Fanuc TP program (LS listing): MOTIONPROBE.LS

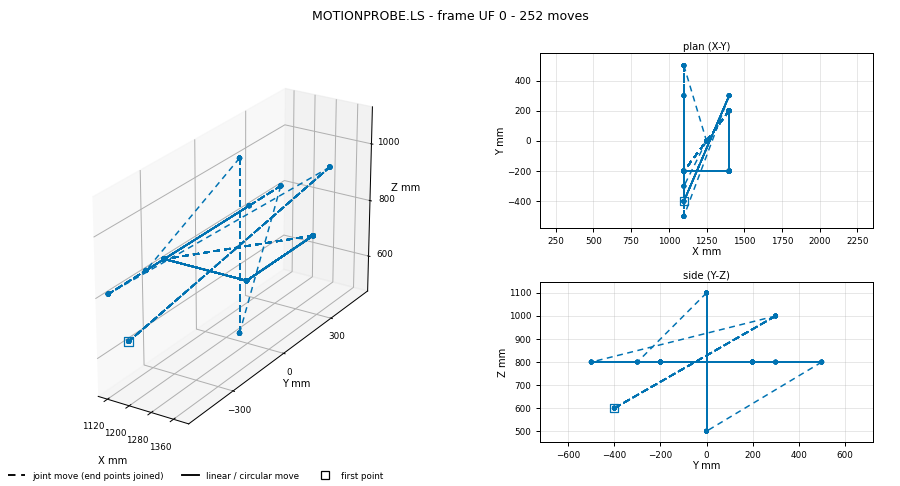
[picture p0: tool path of MOTIONPROBE.LS in frame UF 0, 252 of 252 moves have a stored position in this frame; points joined in program order, loops and branches not executed]
/PROG  MOTIONPROBE
/ATTR
OWNER		= MNEDITOR;
COMMENT		= "motion probe";
PROG_SIZE	= 0;
CREATE		= DATE 26-01-01  TIME 00:00:00;
MODIFIED	= DATE 26-01-01  TIME 00:00:00;
FILE_NAME	= ;
VERSION		= 0;
LINE_COUNT	= 737;
MEMORY_SIZE	= 0;
PROTECT		= READ_WRITE;
TCD:  STACK_SIZE	= 0,
      TASK_PRIORITY	= 50,
      TIME_SLICE	= 0,
      BUSY_LAMP_OFF	= 0,
      ABORT_REQUEST	= 0,
      PAUSE_REQUEST	= 0;
DEFAULT_GROUP	= 1,*,*,*,*;
CONTROL_CODE	= 00000000 00000000;
/MN
   1:  !CrossArm motion probe ;
   2:  PR[20]=P[12]    ;
   3:  UTOOL[1]=PR[20] ;
   4:  UFRAME_NUM=0 ;
   5:  UTOOL_NUM=1 ;
   6:  !joint 5% ;
   7:J P[6] 30% FINE    ;
   8:  TIMER[1]=RESET ;
   9:  TIMER[1]=START ;
  10:J P[7] 5% FINE    ;
  11:  TIMER[1]=STOP ;
  12:  R[101]=TIMER[1]    ;
  13:  !joint 10% ;
  14:J P[6] 30% FINE    ;
  15:  TIMER[1]=RESET ;
  16:  TIMER[1]=START ;
  17:J P[7] 10% FINE    ;
  18:  TIMER[1]=STOP ;
  19:  R[102]=TIMER[1]    ;
  20:  !joint 15% ;
  21:J P[6] 30% FINE    ;
  22:  TIMER[1]=RESET ;
  23:  TIMER[1]=START ;
  24:J P[7] 15% FINE    ;
  25:  TIMER[1]=STOP ;
  26:  R[103]=TIMER[1]    ;
  27:  !joint 20% ;
  28:J P[6] 30% FINE    ;
  29:  TIMER[1]=RESET ;
  30:  TIMER[1]=START ;
  31:J P[7] 20% FINE    ;
  32:  TIMER[1]=STOP ;
  33:  R[104]=TIMER[1]    ;
  34:  !joint 25% ;
  35:J P[6] 30% FINE    ;
  36:  TIMER[1]=RESET ;
  37:  TIMER[1]=START ;
  38:J P[7] 25% FINE    ;
  39:  TIMER[1]=STOP ;
  40:  R[105]=TIMER[1]    ;
  41:  !joint 30% ;
  42:J P[6] 30% FINE    ;
  43:  TIMER[1]=RESET ;
  44:  TIMER[1]=START ;
  45:J P[7] 30% FINE    ;
  46:  TIMER[1]=STOP ;
  47:  R[106]=TIMER[1]    ;
  48:  !joint 40% ;
  49:J P[6] 30% FINE    ;
  50:  TIMER[1]=RESET ;
  51:  TIMER[1]=START ;
  52:J P[7] 40% FINE    ;
  53:  TIMER[1]=STOP ;
  54:  R[107]=TIMER[1]    ;
  55:  !joint 50% ;
  56:J P[6] 30% FINE    ;
  57:  TIMER[1]=RESET ;
  58:  TIMER[1]=START ;
  59:J P[7] 50% FINE    ;
  60:  TIMER[1]=STOP ;
  61:  R[108]=TIMER[1]    ;
  62:  !joint 70% ;
  63:J P[6] 30% FINE    ;
  64:  TIMER[1]=RESET ;
  65:  TIMER[1]=START ;
  66:J P[7] 70% FINE    ;
  67:  TIMER[1]=STOP ;
  68:  R[109]=TIMER[1]    ;
  69:  !joint 100% ;
  70:J P[6] 30% FINE    ;
  71:  TIMER[1]=RESET ;
  72:  TIMER[1]=START ;
  73:J P[7] 100% FINE    ;
  74:  TIMER[1]=STOP ;
  75:  R[110]=TIMER[1]    ;
  76:  !swing 5% ;
  77:J P[8] 30% FINE    ;
  78:  TIMER[1]=RESET ;
  79:  TIMER[1]=START ;
  80:J P[9] 5% FINE    ;
  81:  TIMER[1]=STOP ;
  82:  R[111]=TIMER[1]    ;
  83:  !swing 10% ;
  84:J P[8] 30% FINE    ;
  85:  TIMER[1]=RESET ;
  86:  TIMER[1]=START ;
  87:J P[9] 10% FINE    ;
  88:  TIMER[1]=STOP ;
  89:  R[112]=TIMER[1]    ;
  90:  !swing 15% ;
  91:J P[8] 30% FINE    ;
  92:  TIMER[1]=RESET ;
  93:  TIMER[1]=START ;
  94:J P[9] 15% FINE    ;
  95:  TIMER[1]=STOP ;
  96:  R[113]=TIMER[1]    ;
  97:  !swing 20% ;
  98:J P[8] 30% FINE    ;
  99:  TIMER[1]=RESET ;
 100:  TIMER[1]=START ;
 101:J P[9] 20% FINE    ;
 102:  TIMER[1]=STOP ;
 103:  R[114]=TIMER[1]    ;
 104:  !swing 25% ;
 105:J P[8] 30% FINE    ;
 106:  TIMER[1]=RESET ;
 107:  TIMER[1]=START ;
 108:J P[9] 25% FINE    ;
 109:  TIMER[1]=STOP ;
 110:  R[115]=TIMER[1]    ;
 111:  !swing 30% ;
 112:J P[8] 30% FINE    ;
 113:  TIMER[1]=RESET ;
 114:  TIMER[1]=START ;
 115:J P[9] 30% FINE    ;
 116:  TIMER[1]=STOP ;
 117:  R[116]=TIMER[1]    ;
 118:  !swing 40% ;
 119:J P[8] 30% FINE    ;
 120:  TIMER[1]=RESET ;
 121:  TIMER[1]=START ;
 122:J P[9] 40% FINE    ;
 123:  TIMER[1]=STOP ;
 124:  R[117]=TIMER[1]    ;
 125:  !swing 50% ;
 126:J P[8] 30% FINE    ;
 127:  TIMER[1]=RESET ;
 128:  TIMER[1]=START ;
 129:J P[9] 50% FINE    ;
 130:  TIMER[1]=STOP ;
 131:  R[118]=TIMER[1]    ;
 132:  !swing 70% ;
 133:J P[8] 30% FINE    ;
 134:  TIMER[1]=RESET ;
 135:  TIMER[1]=START ;
 136:J P[9] 70% FINE    ;
 137:  TIMER[1]=STOP ;
 138:  R[119]=TIMER[1]    ;
 139:  !swing 100% ;
 140:J P[8] 30% FINE    ;
 141:  TIMER[1]=RESET ;
 142:  TIMER[1]=START ;
 143:J P[9] 100% FINE    ;
 144:  TIMER[1]=STOP ;
 145:  R[120]=TIMER[1]    ;
 146:  !rise 5% ;
 147:J P[10] 30% FINE    ;
 148:  TIMER[1]=RESET ;
 149:  TIMER[1]=START ;
 150:J P[11] 5% FINE    ;
 151:  TIMER[1]=STOP ;
 152:  R[121]=TIMER[1]    ;
 153:  !rise 10% ;
 154:J P[10] 30% FINE    ;
 155:  TIMER[1]=RESET ;
 156:  TIMER[1]=START ;
 157:J P[11] 10% FINE    ;
 158:  TIMER[1]=STOP ;
 159:  R[122]=TIMER[1]    ;
 160:  !rise 15% ;
 161:J P[10] 30% FINE    ;
 162:  TIMER[1]=RESET ;
 163:  TIMER[1]=START ;
 164:J P[11] 15% FINE    ;
 165:  TIMER[1]=STOP ;
 166:  R[123]=TIMER[1]    ;
 167:  !rise 20% ;
 168:J P[10] 30% FINE    ;
 169:  TIMER[1]=RESET ;
 170:  TIMER[1]=START ;
 171:J P[11] 20% FINE    ;
 172:  TIMER[1]=STOP ;
 173:  R[124]=TIMER[1]    ;
 174:  !rise 25% ;
 175:J P[10] 30% FINE    ;
 176:  TIMER[1]=RESET ;
 177:  TIMER[1]=START ;
 178:J P[11] 25% FINE    ;
 179:  TIMER[1]=STOP ;
 180:  R[125]=TIMER[1]    ;
 181:  !rise 30% ;
 182:J P[10] 30% FINE    ;
 183:  TIMER[1]=RESET ;
 184:  TIMER[1]=START ;
 185:J P[11] 30% FINE    ;
 186:  TIMER[1]=STOP ;
 187:  R[126]=TIMER[1]    ;
 188:  !rise 40% ;
 189:J P[10] 30% FINE    ;
 190:  TIMER[1]=RESET ;
 191:  TIMER[1]=START ;
 192:J P[11] 40% FINE    ;
 193:  TIMER[1]=STOP ;
 194:  R[127]=TIMER[1]    ;
 195:  !rise 50% ;
 196:J P[10] 30% FINE    ;
 197:  TIMER[1]=RESET ;
 198:  TIMER[1]=START ;
 199:J P[11] 50% FINE    ;
 200:  TIMER[1]=STOP ;
 201:  R[128]=TIMER[1]    ;
 202:  !rise 70% ;
 203:J P[10] 30% FINE    ;
 204:  TIMER[1]=RESET ;
 205:  TIMER[1]=START ;
 206:J P[11] 70% FINE    ;
 207:  TIMER[1]=STOP ;
 208:  R[129]=TIMER[1]    ;
 209:  !rise 100% ;
 210:J P[10] 30% FINE    ;
 211:  TIMER[1]=RESET ;
 212:  TIMER[1]=START ;
 213:J P[11] 100% FINE    ;
 214:  TIMER[1]=STOP ;
 215:  R[130]=TIMER[1]    ;
 216:  !linear 100mm/sec ;
 217:J P[4] 30% FINE    ;
 218:  TIMER[1]=RESET ;
 219:  TIMER[1]=START ;
 220:L P[5] 100mm/sec FINE    ;
 221:  TIMER[1]=STOP ;
 222:  R[131]=TIMER[1]    ;
 223:  !linear 200mm/sec ;
 224:J P[4] 30% FINE    ;
 225:  TIMER[1]=RESET ;
 226:  TIMER[1]=START ;
 227:L P[5] 200mm/sec FINE    ;
 228:  TIMER[1]=STOP ;
 229:  R[132]=TIMER[1]    ;
 230:  !linear 500mm/sec ;
 231:J P[4] 30% FINE    ;
 232:  TIMER[1]=RESET ;
 233:  TIMER[1]=START ;
 234:L P[5] 500mm/sec FINE    ;
 235:  TIMER[1]=STOP ;
 236:  R[133]=TIMER[1]    ;
 237:  !linear 1000mm/sec ;
 238:J P[4] 30% FINE    ;
 239:  TIMER[1]=RESET ;
 240:  TIMER[1]=START ;
 241:L P[5] 1000mm/sec FINE    ;
 242:  TIMER[1]=STOP ;
 243:  R[134]=TIMER[1]    ;
 244:  !linear 1500mm/sec ;
 245:J P[4] 30% FINE    ;
 246:  TIMER[1]=RESET ;
 247:  TIMER[1]=START ;
 248:L P[5] 1500mm/sec FINE    ;
 249:  TIMER[1]=STOP ;
 250:  R[135]=TIMER[1]    ;
 251:  !linear 2000mm/sec ;
 252:J P[4] 30% FINE    ;
 253:  TIMER[1]=RESET ;
 254:  TIMER[1]=START ;
 255:L P[5] 2000mm/sec FINE    ;
 256:  TIMER[1]=STOP ;
 257:  R[136]=TIMER[1]    ;
 258:  !corner 200mm/sec FINE ;
 259:J P[1] 30% FINE    ;
 260:  TIMER[1]=RESET ;
 261:  TIMER[1]=START ;
 262:L P[2] 200mm/sec FINE    ;
 263:L P[3] 200mm/sec FINE    ;
 264:  TIMER[1]=STOP ;
 265:  R[137]=TIMER[1]    ;
 266:  !corner 200mm/sec CNT0 ;
 267:J P[1] 30% FINE    ;
 268:  TIMER[1]=RESET ;
 269:  TIMER[1]=START ;
 270:L P[2] 200mm/sec CNT0    ;
 271:L P[3] 200mm/sec FINE    ;
 272:  TIMER[1]=STOP ;
 273:  R[138]=TIMER[1]    ;
 274:  !corner 200mm/sec CNT10 ;
 275:J P[1] 30% FINE    ;
 276:  TIMER[1]=RESET ;
 277:  TIMER[1]=START ;
 278:L P[2] 200mm/sec CNT10    ;
 279:L P[3] 200mm/sec FINE    ;
 280:  TIMER[1]=STOP ;
 281:  R[139]=TIMER[1]    ;
 282:  !corner 200mm/sec CNT20 ;
 283:J P[1] 30% FINE    ;
 284:  TIMER[1]=RESET ;
 285:  TIMER[1]=START ;
 286:L P[2] 200mm/sec CNT20    ;
 287:L P[3] 200mm/sec FINE    ;
 288:  TIMER[1]=STOP ;
 289:  R[140]=TIMER[1]    ;
 290:  !corner 200mm/sec CNT30 ;
 291:J P[1] 30% FINE    ;
 292:  TIMER[1]=RESET ;
 293:  TIMER[1]=START ;
 294:L P[2] 200mm/sec CNT30    ;
 295:L P[3] 200mm/sec FINE    ;
 296:  TIMER[1]=STOP ;
 297:  R[141]=TIMER[1]    ;
 298:  !corner 200mm/sec CNT40 ;
 299:J P[1] 30% FINE    ;
 300:  TIMER[1]=RESET ;
 301:  TIMER[1]=START ;
 302:L P[2] 200mm/sec CNT40    ;
 303:L P[3] 200mm/sec FINE    ;
 304:  TIMER[1]=STOP ;
 305:  R[142]=TIMER[1]    ;
 306:  !corner 200mm/sec CNT50 ;
 307:J P[1] 30% FINE    ;
 308:  TIMER[1]=RESET ;
 309:  TIMER[1]=START ;
 310:L P[2] 200mm/sec CNT50    ;
 311:L P[3] 200mm/sec FINE    ;
 312:  TIMER[1]=STOP ;
 313:  R[143]=TIMER[1]    ;
 314:  !corner 200mm/sec CNT60 ;
 315:J P[1] 30% FINE    ;
 316:  TIMER[1]=RESET ;
 317:  TIMER[1]=START ;
 318:L P[2] 200mm/sec CNT60    ;
 319:L P[3] 200mm/sec FINE    ;
 320:  TIMER[1]=STOP ;
 321:  R[144]=TIMER[1]    ;
 322:  !corner 200mm/sec CNT70 ;
 323:J P[1] 30% FINE    ;
 324:  TIMER[1]=RESET ;
 325:  TIMER[1]=START ;
 326:L P[2] 200mm/sec CNT70    ;
 327:L P[3] 200mm/sec FINE    ;
 328:  TIMER[1]=STOP ;
 329:  R[145]=TIMER[1]    ;
 330:  !corner 200mm/sec CNT80 ;
 331:J P[1] 30% FINE    ;
 332:  TIMER[1]=RESET ;
 333:  TIMER[1]=START ;
 334:L P[2] 200mm/sec CNT80    ;
 335:L P[3] 200mm/sec FINE    ;
 336:  TIMER[1]=STOP ;
 337:  R[146]=TIMER[1]    ;
 338:  !corner 200mm/sec CNT90 ;
 339:J P[1] 30% FINE    ;
 340:  TIMER[1]=RESET ;
 341:  TIMER[1]=START ;
 342:L P[2] 200mm/sec CNT90    ;
 343:L P[3] 200mm/sec FINE    ;
 344:  TIMER[1]=STOP ;
 345:  R[147]=TIMER[1]    ;
 346:  !corner 200mm/sec CNT100 ;
 347:J P[1] 30% FINE    ;
 348:  TIMER[1]=RESET ;
 349:  TIMER[1]=START ;
 350:L P[2] 200mm/sec CNT100    ;
 351:L P[3] 200mm/sec FINE    ;
 352:  TIMER[1]=STOP ;
 353:  R[148]=TIMER[1]    ;
 354:  !corner 500mm/sec FINE ;
 355:J P[1] 30% FINE    ;
 356:  TIMER[1]=RESET ;
 357:  TIMER[1]=START ;
 358:L P[2] 500mm/sec FINE    ;
 359:L P[3] 500mm/sec FINE    ;
 360:  TIMER[1]=STOP ;
 361:  R[149]=TIMER[1]    ;
 362:  !corner 500mm/sec CNT0 ;
 363:J P[1] 30% FINE    ;
 364:  TIMER[1]=RESET ;
 365:  TIMER[1]=START ;
 366:L P[2] 500mm/sec CNT0    ;
 367:L P[3] 500mm/sec FINE    ;
 368:  TIMER[1]=STOP ;
 369:  R[150]=TIMER[1]    ;
 370:  !corner 500mm/sec CNT10 ;
 371:J P[1] 30% FINE    ;
 372:  TIMER[1]=RESET ;
 373:  TIMER[1]=START ;
 374:L P[2] 500mm/sec CNT10    ;
 375:L P[3] 500mm/sec FINE    ;
 376:  TIMER[1]=STOP ;
 377:  R[151]=TIMER[1]    ;
 378:  !corner 500mm/sec CNT20 ;
 379:J P[1] 30% FINE    ;
 380:  TIMER[1]=RESET ;
 381:  TIMER[1]=START ;
 382:L P[2] 500mm/sec CNT20    ;
 383:L P[3] 500mm/sec FINE    ;
 384:  TIMER[1]=STOP ;
 385:  R[152]=TIMER[1]    ;
 386:  !corner 500mm/sec CNT30 ;
 387:J P[1] 30% FINE    ;
 388:  TIMER[1]=RESET ;
 389:  TIMER[1]=START ;
 390:L P[2] 500mm/sec CNT30    ;
 391:L P[3] 500mm/sec FINE    ;
 392:  TIMER[1]=STOP ;
 393:  R[153]=TIMER[1]    ;
 394:  !corner 500mm/sec CNT40 ;
 395:J P[1] 30% FINE    ;
 396:  TIMER[1]=RESET ;
 397:  TIMER[1]=START ;
 398:L P[2] 500mm/sec CNT40    ;
 399:L P[3] 500mm/sec FINE    ;
 400:  TIMER[1]=STOP ;
 401:  R[154]=TIMER[1]    ;
 402:  !corner 500mm/sec CNT50 ;
 403:J P[1] 30% FINE    ;
 404:  TIMER[1]=RESET ;
 405:  TIMER[1]=START ;
 406:L P[2] 500mm/sec CNT50    ;
 407:L P[3] 500mm/sec FINE    ;
 408:  TIMER[1]=STOP ;
 409:  R[155]=TIMER[1]    ;
 410:  !corner 500mm/sec CNT60 ;
 411:J P[1] 30% FINE    ;
 412:  TIMER[1]=RESET ;
 413:  TIMER[1]=START ;
 414:L P[2] 500mm/sec CNT60    ;
 415:L P[3] 500mm/sec FINE    ;
 416:  TIMER[1]=STOP ;
 417:  R[156]=TIMER[1]    ;
 418:  !corner 500mm/sec CNT70 ;
 419:J P[1] 30% FINE    ;
 420:  TIMER[1]=RESET ;
 421:  TIMER[1]=START ;
 422:L P[2] 500mm/sec CNT70    ;
 423:L P[3] 500mm/sec FINE    ;
 424:  TIMER[1]=STOP ;
 425:  R[157]=TIMER[1]    ;
 426:  !corner 500mm/sec CNT80 ;
 427:J P[1] 30% FINE    ;
 428:  TIMER[1]=RESET ;
 429:  TIMER[1]=START ;
 430:L P[2] 500mm/sec CNT80    ;
 431:L P[3] 500mm/sec FINE    ;
 432:  TIMER[1]=STOP ;
 433:  R[158]=TIMER[1]    ;
 434:  !corner 500mm/sec CNT90 ;
 435:J P[1] 30% FINE    ;
 436:  TIMER[1]=RESET ;
 437:  TIMER[1]=START ;
 438:L P[2] 500mm/sec CNT90    ;
 439:L P[3] 500mm/sec FINE    ;
 440:  TIMER[1]=STOP ;
 441:  R[159]=TIMER[1]    ;
 442:  !corner 500mm/sec CNT100 ;
 443:J P[1] 30% FINE    ;
 444:  TIMER[1]=RESET ;
 445:  TIMER[1]=START ;
 446:L P[2] 500mm/sec CNT100    ;
 447:L P[3] 500mm/sec FINE    ;
 448:  TIMER[1]=STOP ;
 449:  R[160]=TIMER[1]    ;
 450:  !corner 1000mm/sec FINE ;
 451:J P[1] 30% FINE    ;
 452:  TIMER[1]=RESET ;
 453:  TIMER[1]=START ;
 454:L P[2] 1000mm/sec FINE    ;
 455:L P[3] 1000mm/sec FINE    ;
 456:  TIMER[1]=STOP ;
 457:  R[161]=TIMER[1]    ;
 458:  !corner 1000mm/sec CNT0 ;
 459:J P[1] 30% FINE    ;
 460:  TIMER[1]=RESET ;
 461:  TIMER[1]=START ;
 462:L P[2] 1000mm/sec CNT0    ;
 463:L P[3] 1000mm/sec FINE    ;
 464:  TIMER[1]=STOP ;
 465:  R[162]=TIMER[1]    ;
 466:  !corner 1000mm/sec CNT10 ;
 467:J P[1] 30% FINE    ;
 468:  TIMER[1]=RESET ;
 469:  TIMER[1]=START ;
 470:L P[2] 1000mm/sec CNT10    ;
 471:L P[3] 1000mm/sec FINE    ;
 472:  TIMER[1]=STOP ;
 473:  R[163]=TIMER[1]    ;
 474:  !corner 1000mm/sec CNT20 ;
 475:J P[1] 30% FINE    ;
 476:  TIMER[1]=RESET ;
 477:  TIMER[1]=START ;
 478:L P[2] 1000mm/sec CNT20    ;
 479:L P[3] 1000mm/sec FINE    ;
 480:  TIMER[1]=STOP ;
 481:  R[164]=TIMER[1]    ;
 482:  !corner 1000mm/sec CNT30 ;
 483:J P[1] 30% FINE    ;
 484:  TIMER[1]=RESET ;
 485:  TIMER[1]=START ;
 486:L P[2] 1000mm/sec CNT30    ;
 487:L P[3] 1000mm/sec FINE    ;
 488:  TIMER[1]=STOP ;
 489:  R[165]=TIMER[1]    ;
 490:  !corner 1000mm/sec CNT40 ;
 491:J P[1] 30% FINE    ;
 492:  TIMER[1]=RESET ;
 493:  TIMER[1]=START ;
 494:L P[2] 1000mm/sec CNT40    ;
 495:L P[3] 1000mm/sec FINE    ;
 496:  TIMER[1]=STOP ;
 497:  R[166]=TIMER[1]    ;
 498:  !corner 1000mm/sec CNT50 ;
 499:J P[1] 30% FINE    ;
 500:  TIMER[1]=RESET ;
 501:  TIMER[1]=START ;
 502:L P[2] 1000mm/sec CNT50    ;
 503:L P[3] 1000mm/sec FINE    ;
 504:  TIMER[1]=STOP ;
 505:  R[167]=TIMER[1]    ;
 506:  !corner 1000mm/sec CNT60 ;
 507:J P[1] 30% FINE    ;
 508:  TIMER[1]=RESET ;
 509:  TIMER[1]=START ;
 510:L P[2] 1000mm/sec CNT60    ;
 511:L P[3] 1000mm/sec FINE    ;
 512:  TIMER[1]=STOP ;
 513:  R[168]=TIMER[1]    ;
 514:  !corner 1000mm/sec CNT70 ;
 515:J P[1] 30% FINE    ;
 516:  TIMER[1]=RESET ;
 517:  TIMER[1]=START ;
 518:L P[2] 1000mm/sec CNT70    ;
 519:L P[3] 1000mm/sec FINE    ;
 520:  TIMER[1]=STOP ;
 521:  R[169]=TIMER[1]    ;
 522:  !corner 1000mm/sec CNT80 ;
 523:J P[1] 30% FINE    ;
 524:  TIMER[1]=RESET ;
 525:  TIMER[1]=START ;
 526:L P[2] 1000mm/sec CNT80    ;
 527:L P[3] 1000mm/sec FINE    ;
 528:  TIMER[1]=STOP ;
 529:  R[170]=TIMER[1]    ;
 530:  !corner 1000mm/sec CNT90 ;
 531:J P[1] 30% FINE    ;
 532:  TIMER[1]=RESET ;
 533:  TIMER[1]=START ;
 534:L P[2] 1000mm/sec CNT90    ;
 535:L P[3] 1000mm/sec FINE    ;
 536:  TIMER[1]=STOP ;
 537:  R[171]=TIMER[1]    ;
 538:  !corner 1000mm/sec CNT100 ;
 539:J P[1] 30% FINE    ;
 540:  TIMER[1]=RESET ;
 541:  TIMER[1]=START ;
 542:L P[2] 1000mm/sec CNT100    ;
 543:L P[3] 1000mm/sec FINE    ;
 544:  TIMER[1]=STOP ;
 545:  R[172]=TIMER[1]    ;
 546:  !jcorner 9% FINE ;
 547:J P[1] 30% FINE    ;
 548:  TIMER[1]=RESET ;
 549:  TIMER[1]=START ;
 550:J P[2] 9% FINE    ;
 551:J P[3] 9% FINE    ;
 552:  TIMER[1]=STOP ;
 553:  R[173]=TIMER[1]    ;
 554:  !jcorner 9% CNT0 ;
 555:J P[1] 30% FINE    ;
 556:  TIMER[1]=RESET ;
 557:  TIMER[1]=START ;
 558:J P[2] 9% CNT0    ;
 559:J P[3] 9% FINE    ;
 560:  TIMER[1]=STOP ;
 561:  R[174]=TIMER[1]    ;
 562:  !jcorner 9% CNT10 ;
 563:J P[1] 30% FINE    ;
 564:  TIMER[1]=RESET ;
 565:  TIMER[1]=START ;
 566:J P[2] 9% CNT10    ;
 567:J P[3] 9% FINE    ;
 568:  TIMER[1]=STOP ;
 569:  R[175]=TIMER[1]    ;
 570:  !jcorner 9% CNT20 ;
 571:J P[1] 30% FINE    ;
 572:  TIMER[1]=RESET ;
 573:  TIMER[1]=START ;
 574:J P[2] 9% CNT20    ;
 575:J P[3] 9% FINE    ;
 576:  TIMER[1]=STOP ;
 577:  R[176]=TIMER[1]    ;
 578:  !jcorner 9% CNT30 ;
 579:J P[1] 30% FINE    ;
 580:  TIMER[1]=RESET ;
 581:  TIMER[1]=START ;
 582:J P[2] 9% CNT30    ;
 583:J P[3] 9% FINE    ;
 584:  TIMER[1]=STOP ;
 585:  R[177]=TIMER[1]    ;
 586:  !jcorner 9% CNT40 ;
 587:J P[1] 30% FINE    ;
 588:  TIMER[1]=RESET ;
 589:  TIMER[1]=START ;
 590:J P[2] 9% CNT40    ;
 591:J P[3] 9% FINE    ;
 592:  TIMER[1]=STOP ;
 593:  R[178]=TIMER[1]    ;
 594:  !jcorner 9% CNT50 ;
 595:J P[1] 30% FINE    ;
 596:  TIMER[1]=RESET ;
 597:  TIMER[1]=START ;
 598:J P[2] 9% CNT50    ;
 599:J P[3] 9% FINE    ;
 600:  TIMER[1]=STOP ;
 601:  R[179]=TIMER[1]    ;
 602:  !jcorner 9% CNT60 ;
 603:J P[1] 30% FINE    ;
 604:  TIMER[1]=RESET ;
 605:  TIMER[1]=START ;
 606:J P[2] 9% CNT60    ;
 607:J P[3] 9% FINE    ;
 608:  TIMER[1]=STOP ;
 609:  R[180]=TIMER[1]    ;
 610:  !jcorner 9% CNT70 ;
 611:J P[1] 30% FINE    ;
 612:  TIMER[1]=RESET ;
 613:  TIMER[1]=START ;
 614:J P[2] 9% CNT70    ;
 615:J P[3] 9% FINE    ;
 616:  TIMER[1]=STOP ;
 617:  R[181]=TIMER[1]    ;
 618:  !jcorner 9% CNT80 ;
 619:J P[1] 30% FINE    ;
 620:  TIMER[1]=RESET ;
 621:  TIMER[1]=START ;
 622:J P[2] 9% CNT80    ;
 623:J P[3] 9% FINE    ;
 624:  TIMER[1]=STOP ;
 625:  R[182]=TIMER[1]    ;
 626:  !jcorner 9% CNT90 ;
 627:J P[1] 30% FINE    ;
 628:  TIMER[1]=RESET ;
 629:  TIMER[1]=START ;
 630:J P[2] 9% CNT90    ;
 631:J P[3] 9% FINE    ;
 632:  TIMER[1]=STOP ;
 633:  R[183]=TIMER[1]    ;
 634:  !jcorner 9% CNT100 ;
 635:J P[1] 30% FINE    ;
 636:  TIMER[1]=RESET ;
 637:  TIMER[1]=START ;
 638:J P[2] 9% CNT100    ;
 639:J P[3] 9% FINE    ;
 640:  TIMER[1]=STOP ;
 641:  R[184]=TIMER[1]    ;
 642:  !jcorner 19% FINE ;
 643:J P[1] 30% FINE    ;
 644:  TIMER[1]=RESET ;
 645:  TIMER[1]=START ;
 646:J P[2] 19% FINE    ;
 647:J P[3] 19% FINE    ;
 648:  TIMER[1]=STOP ;
 649:  R[185]=TIMER[1]    ;
 650:  !jcorner 19% CNT0 ;
 651:J P[1] 30% FINE    ;
 652:  TIMER[1]=RESET ;
 653:  TIMER[1]=START ;
 654:J P[2] 19% CNT0    ;
 655:J P[3] 19% FINE    ;
 656:  TIMER[1]=STOP ;
 657:  R[186]=TIMER[1]    ;
 658:  !jcorner 19% CNT10 ;
 659:J P[1] 30% FINE    ;
 660:  TIMER[1]=RESET ;
 661:  TIMER[1]=START ;
 662:J P[2] 19% CNT10    ;
 663:J P[3] 19% FINE    ;
 664:  TIMER[1]=STOP ;
 665:  R[187]=TIMER[1]    ;
 666:  !jcorner 19% CNT20 ;
 667:J P[1] 30% FINE    ;
 668:  TIMER[1]=RESET ;
 669:  TIMER[1]=START ;
 670:J P[2] 19% CNT20    ;
 671:J P[3] 19% FINE    ;
 672:  TIMER[1]=STOP ;
 673:  R[188]=TIMER[1]    ;
 674:  !jcorner 19% CNT30 ;
 675:J P[1] 30% FINE    ;
 676:  TIMER[1]=RESET ;
 677:  TIMER[1]=START ;
 678:J P[2] 19% CNT30    ;
 679:J P[3] 19% FINE    ;
 680:  TIMER[1]=STOP ;
 681:  R[189]=TIMER[1]    ;
 682:  !jcorner 19% CNT40 ;
 683:J P[1] 30% FINE    ;
 684:  TIMER[1]=RESET ;
 685:  TIMER[1]=START ;
 686:J P[2] 19% CNT40    ;
 687:J P[3] 19% FINE    ;
 688:  TIMER[1]=STOP ;
 689:  R[190]=TIMER[1]    ;
 690:  !jcorner 19% CNT50 ;
 691:J P[1] 30% FINE    ;
 692:  TIMER[1]=RESET ;
 693:  TIMER[1]=START ;
 694:J P[2] 19% CNT50    ;
 695:J P[3] 19% FINE    ;
 696:  TIMER[1]=STOP ;
 697:  R[191]=TIMER[1]    ;
 698:  !jcorner 19% CNT60 ;
 699:J P[1] 30% FINE    ;
 700:  TIMER[1]=RESET ;
 701:  TIMER[1]=START ;
 702:J P[2] 19% CNT60    ;
 703:J P[3] 19% FINE    ;
 704:  TIMER[1]=STOP ;
 705:  R[192]=TIMER[1]    ;
 706:  !jcorner 19% CNT70 ;
 707:J P[1] 30% FINE    ;
 708:  TIMER[1]=RESET ;
 709:  TIMER[1]=START ;
 710:J P[2] 19% CNT70    ;
 711:J P[3] 19% FINE    ;
 712:  TIMER[1]=STOP ;
 713:  R[193]=TIMER[1]    ;
 714:  !jcorner 19% CNT80 ;
 715:J P[1] 30% FINE    ;
 716:  TIMER[1]=RESET ;
 717:  TIMER[1]=START ;
 718:J P[2] 19% CNT80    ;
 719:J P[3] 19% FINE    ;
 720:  TIMER[1]=STOP ;
 721:  R[194]=TIMER[1]    ;
 722:  !jcorner 19% CNT90 ;
 723:J P[1] 30% FINE    ;
 724:  TIMER[1]=RESET ;
 725:  TIMER[1]=START ;
 726:J P[2] 19% CNT90    ;
 727:J P[3] 19% FINE    ;
 728:  TIMER[1]=STOP ;
 729:  R[195]=TIMER[1]    ;
 730:  !jcorner 19% CNT100 ;
 731:J P[1] 30% FINE    ;
 732:  TIMER[1]=RESET ;
 733:  TIMER[1]=START ;
 734:J P[2] 19% CNT100    ;
 735:J P[3] 19% FINE    ;
 736:  TIMER[1]=STOP ;
 737:  R[196]=TIMER[1]    ;
/POS
P[1]{
   GP1:
	UF : 0, UT : 1,		CONFIG : 'N U T, 0, 0, 0',
	X =  1100.000  mm,	Y =  -200.000  mm,	Z =   800.000  mm,
	W =   180.000 deg,	P =     0.000 deg,	R =   135.000 deg
};
P[2]{
   GP1:
	UF : 0, UT : 1,		CONFIG : 'N U T, 0, 0, 0',
	X =  1400.000  mm,	Y =  -200.000  mm,	Z =   800.000  mm,
	W =   180.000 deg,	P =     0.000 deg,	R =   135.000 deg
};
P[3]{
   GP1:
	UF : 0, UT : 1,		CONFIG : 'N U T, 0, 0, 0',
	X =  1400.000  mm,	Y =   200.000  mm,	Z =   800.000  mm,
	W =   180.000 deg,	P =     0.000 deg,	R =   135.000 deg
};
P[4]{
   GP1:
	UF : 0, UT : 1,		CONFIG : 'N U T, 0, 0, 0',
	X =  1100.000  mm,	Y =  -300.000  mm,	Z =   800.000  mm,
	W =   180.000 deg,	P =     0.000 deg,	R =   135.000 deg
};
P[5]{
   GP1:
	UF : 0, UT : 1,		CONFIG : 'N U T, 0, 0, 0',
	X =  1100.000  mm,	Y =   300.000  mm,	Z =   800.000  mm,
	W =   180.000 deg,	P =     0.000 deg,	R =   135.000 deg
};
P[6]{
   GP1:
	UF : 0, UT : 1,		CONFIG : 'N U T, 0, 0, 0',
	X =  1100.000  mm,	Y =  -400.000  mm,	Z =   600.000  mm,
	W =   180.000 deg,	P =     0.000 deg,	R =   135.000 deg
};
P[7]{
   GP1:
	UF : 0, UT : 1,		CONFIG : 'N U T, 0, 0, 0',
	X =  1400.000  mm,	Y =   300.000  mm,	Z =  1000.000  mm,
	W =   180.000 deg,	P =     0.000 deg,	R =   135.000 deg
};
P[8]{
   GP1:
	UF : 0, UT : 1,		CONFIG : 'N U T, 0, 0, 0',
	X =  1100.000  mm,	Y =  -500.000  mm,	Z =   800.000  mm,
	W =   180.000 deg,	P =     0.000 deg,	R =   135.000 deg
};
P[9]{
   GP1:
	UF : 0, UT : 1,		CONFIG : 'N U T, 0, 0, 0',
	X =  1100.000  mm,	Y =   500.000  mm,	Z =   800.000  mm,
	W =   180.000 deg,	P =     0.000 deg,	R =   135.000 deg
};
P[10]{
   GP1:
	UF : 0, UT : 1,		CONFIG : 'N U T, 0, 0, 0',
	X =  1250.000  mm,	Y =     0.000  mm,	Z =   500.000  mm,
	W =   180.000 deg,	P =     0.000 deg,	R =   135.000 deg
};
P[11]{
   GP1:
	UF : 0, UT : 1,		CONFIG : 'N U T, 0, 0, 0',
	X =  1250.000  mm,	Y =     0.000  mm,	Z =  1100.000  mm,
	W =   180.000 deg,	P =     0.000 deg,	R =   135.000 deg
};
P[12]{
   GP1:
	UF : 0, UT : 1,		CONFIG : 'N U T, 0, 0, 0',
	X =     0.000  mm,	Y =     0.000  mm,	Z =     0.000  mm,
	W =     0.000 deg,	P =     0.000 deg,	R =     0.000 deg
};
/END
